{attribute 'no_explicit_call' := 'do not call this FB directly'}{attribute 'enable_dynamic_creation'}
FUNCTION_BLOCK FINAL BoolDisplayNode EXTENDS Node
VAR
	in : _BOOL(FALSE);
	display : _BOOL(FALSE);
END_VAR

METHOD PUBLIC Clone : I_Node
VAR
	pointerToNode : POINTER TO Node_Display_BOOL;
END_VAR
pointerToNode := __NEW(Node_Display_BOOL);
Clone := pointerToNode^;
END_METHOD

METHOD FB_init : BOOL
VAR_INPUT
	bInitRetains : BOOL; // if TRUE, the retain variables are initialized (warm start / cold start)
	bInCopyCode : BOOL;  // if TRUE, the instance afterwards gets moved into the copy code (online change)
END_VAR
InputPorts.AddDataAsInputPort('in', in);
Contents.AddDataAsContent('display', display);
END_METHOD

METHOD PROTECTED OnExecute : HRESULT
display.Value := in.Value;
END_METHOD

END_FUNCTION_BLOCK

(* stored: Version 1.1.0.1, ProductVersion 3.1.4024.12
   POU BoolDisplayNode: Id {0f08307d-4041-4da5-a467-5b06e7eedf33}, SpecialFunc None
   Folder Constructor: Id {227aa244-3e7a-4525-bac6-987f3cb4f2f0}
   Method Clone: Id {becf0f39-df3c-403f-9972-d66a56950b8c}
   Method FB_init: Id {e4cb0d0b-c40f-40c5-b63b-f9237053b3c1}
   Method OnExecute: Id {2fac624a-eb27-478f-8639-998a4165478e} *)
